TYPE FILE_PATH_DATA :
STRUCT
	DRIVE : STRING(3);
	DIRECTORY : STRING(STRING_LENGTH);
	FILENAME : STRING;
END_STRUCT
END_TYPE

(* stored: Version 1.1.0.1, ProductVersion 3.1.4022.7
   DUT FILE_PATH_DATA: Id {c84fbfd8-d07c-4e8a-a640-ef2c25da633d} *)
